// TIA Portal V17 export
// export: Created 2026-04-13T11:12:42.0985192Z, ExportSetting WithDefaults, DisplayName Totally Integrated Automation Portal, DisplayVersion V17 Update 4, DisplayName TIA Portal Openness, DisplayVersion V17 Update 4, DisplayName TIA Portal Version Control Interface, DisplayVersion V17, DisplayName SINAMICS Startdrive Advanced, DisplayVersion V17, DisplayName SINAMICS Startdrive G130, G150, S120, S150, SINAMICS MV, S210, DisplayVersion V17, DisplayName SINAMICS Startdrive G110M, G120, G120C, G120D, G120P, G115D, DisplayVersion V17, DisplayName STEP 7 Professional, DisplayVersion V17 Update 4, DisplayName STEP 7 Safety, DisplayVersion V17, DisplayName WinCC Professional, DisplayVersion V17 Update 4
FUNCTION_BLOCK "自动流程"   // FB82, SCL
{ S7_Optimized_Access := 'TRUE' }
VERSION : 0.1
// stored: AutoNumber true, IsIECCheckEnabled false, IsRetainMemResEnabled false, MemoryReserve 100, SetENOAutomatically false, UDAEnableTagReadback false
   VAR
      execute : Bool;
      stepmode : Bool;
      stepsignal : Bool;
      stepsignalrise : Bool;
      stepsignallast : Bool;
      "step" : Int;
      nextstep : Int;
      "1号cmd" : Bool;
      "1号pos" : Bool;
      "1号homecmd" : Bool;
      "1号homepos" : Bool;
      "2号cmd" : Bool;
      "2号pos" : Bool;
      "2号homecmd" : Bool;
      "2号homepos" : Bool;
   END_VAR
BEGIN
   IF #execute THEN
       CASE #step OF
           0:
               #"1号cmd" := 1;
               IF #"1号pos" THEN
                   #"1号cmd" := 0;
                   #nextstep := 10;
               END_IF;
               ;
           10:
               #"2号cmd" := 1;
               IF #"2号pos" THEN
                   #"2号cmd" := 0;
                   #nextstep := 20;
               END_IF;
               ;
           20:
               #"2号homecmd" := 1;
               IF #"2号homepos" THEN
                   #"2号homecmd" := 0;
                   #nextstep := 30;
               END_IF;
               ;
           30:
               #"1号homecmd" := 1;
               IF #"1号homepos" THEN
                   #"1号homecmd" := 0;
                   #nextstep := 40;
               END_IF;
           ELSE
               ;
       END_CASE;

       #stepsignalrise := #stepsignal AND NOT #stepsignallast;
       #stepsignallast := #stepsignal;
       IF NOT #stepmode OR (#stepmode AND #stepsignalrise) THEN
           #step := #nextstep;
       END_IF;
   ELSE
       #step := 0;
   END_IF;
END_FUNCTION_BLOCK
